FUNCTION_BLOCK B_SECCOM_CONTROLREMOTO (* Basic Function Block Type *)
  (* Standard: 61499-2 *)
  (* Version 0.0, 2015-12-09, 4DIAC-IDE, 4DIAC-Consortium *)
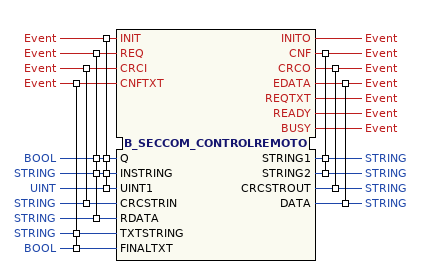
  EVENT_INPUT
    INIT WITH Q, UINT1, INSTRING; (* Initialization Request *)
    REQ WITH Q, INSTRING, RDATA; (* Normal Execution Request *)
    CRCI WITH CRCSTRIN;
    CNFTXT WITH TXTSTRING, FINALTXT;
  END_EVENT
  EVENT_OUTPUT
    INITO; (* Initialization Confirm *)
    CNF WITH STRING1, STRING2; (* Execution Confirmation *)
    CRCO WITH CRCSTROUT;
    EDATA WITH DATA;
    REQTXT;
    READY;
    BUSY;
  END_EVENT
  VAR_INPUT
    Q : BOOL; (* Input event qualifier *)
    INSTRING : STRING;
    UINT1 : UINT;
    CRCSTRIN : STRING;
    RDATA : STRING;
    TXTSTRING : STRING;
    FINALTXT : BOOL;
  END_VAR
  VAR_OUTPUT
    STRING1 : STRING;
    STRING2 : STRING;
    CRCSTROUT : STRING;
    DATA : STRING;
  END_VAR
  VAR
    STRSUB1 : STRING; (* Internal Variable *)
    STRSUB2 : STRING; (* Internal Variable *)
    STRSUB3 : STRING; (* Internal Variable *)
    INITCONTROL : BOOL := FALSE; (* Internal Variable *)
    UINTCPY : UINT := 0; (* Internal Variable *)
    LASTDLE : STRING; (* Internal Variable *)
    STRINGSPACE : STRING; (* Internal Variable *)
    SPACEINT : INT := 0; (* Internal Variable *)
    AUXINT1 : INT := 0; (* Internal Variable *)
    INTERNALVAR2 : BOOL; (* Internal Variable *)
  END_VAR
  EC_STATES
    START;
    State1 : start -> BUSY; (* Initial State *)
    SIMULACIONTECLADO : ST0 -> CNF;
    EJECUCIONPROGRAMA : EP0 -> CNF;
    PETICIONERRORES : PE0 -> CNF;
    LECTURAEJES : ST0 -> CNF;
    INFORMETIPO : ST0 -> CNF;
    ST1 : ST1 -> CRCO;
    ST2 : ST2 -> CNF;
    Exit_ST : -> READY;
    ST3 : ST3 -> CNF;
    ST4 : ST4 -> CNF;
    ST5 : ST5 -> CNF;
    INFOREESTADO : IE0 -> CNF;
    IE1 : IE1 -> CNF;
    IE2 : IE2 -> CNF;
    IE3 : IE3 -> CNF;
    IE4 : IE40 -> EDATA, IE4 -> CNF;
    Exit_IE : -> READY;
    InitEP : INIT -> CNF;
    InitPE : INIT -> CNF;
    Init_ST : INIT -> CNF;
    Init_LE : INIT -> CNF;
    Init_IT : INIT -> CNF;
    Init_IE : INIT -> CNF;
    PE1 : PE1 -> CRCO;
    PE2 : PE2 -> CNF;
    Exit_PE : -> READY;
    PE3 : PE3 -> CNF;
    PE4 : PE4 -> CNF;
    PE5 : PE50 -> EDATA, PE5 -> CNF;
    Exit_IT : -> READY;
    IT1 : IT1 -> CRCO;
    IT2 : ST2 -> CNF;
    IT3 : ST3 -> CNF;
    IT4 : ST4 -> CNF;
    IT5 : IT50 -> EDATA, ST5 -> CNF;
    Exit_LE : -> READY;
    LE1 : LE1 -> CRCO;
    LE2 : ST2 -> CNF;
    LE3 : ST3 -> CNF;
    LE4 : ST4 -> CNF;
    LE5 : LE50 -> EDATA, ST5 -> CNF;
    CARGAPROGRAMA : IE0 -> CNF;
    Exit_CP : -> READY;
    Init_CP : INIT -> CNF;
    CP1 : CP1 -> CRCO;
    CP4 : CP4 -> CRCO;
    CP2 : CP2 -> CNF;
    CP3 : -> REQTXT;
    CP6 : CP6 -> CNF;
    CP5 : CP5 -> CNF;
    EP1 : EP1 -> CRCO;
    EP2 : PE2 -> CNF;
    EP3 : PE3 -> CNF;
    Exit_PE_1 : -> READY;
    EP4 : PE4 -> CNF;
    EP5 : PE50 -> EDATA, PE5 -> CNF;
  END_STATES
  EC_TRANSITIONS
    SIMULACIONTECLADO TO ST1 := REQ&Q;
    ST1 TO ST2 := CRCI;
    SIMULACIONTECLADO TO Exit_ST := REQ&NOT Q;
    ST2 TO ST3 := REQ&Q;
    ST2 TO Exit_ST := REQ&NOT Q;
    ST3 TO ST4 := REQ&Q;
    ST4 TO ST5 := REQ&Q;
    ST3 TO Exit_ST := REQ&NOT Q;
    ST4 TO Exit_ST := REQ&NOT Q;
    ST5 TO Exit_ST := 1;
    INFOREESTADO TO IE1 := REQ&Q;
    IE1 TO IE2 := REQ&Q;
    IE2 TO IE3 := REQ&Q;
    IE3 TO IE4 := REQ&Q;
    INFOREESTADO TO Exit_IE := REQ&NOT Q;
    IE1 TO Exit_IE := REQ&NOT Q;
    IE2 TO Exit_IE := REQ&NOT Q;
    IE3 TO Exit_IE := REQ&NOT Q;
    IE4 TO Exit_IE := 1;
    State1 TO InitEP := UINTCPY=0 & INITCONTROL;
    InitEP TO EJECUCIONPROGRAMA := REQ&Q;
    InitPE TO PETICIONERRORES := REQ&Q;
    State1 TO InitPE := UINTCPY=1 & INITCONTROL;
    State1 TO Init_ST := UINTCPY=2 & INITCONTROL;
    State1 TO Init_LE := UINTCPY=3 & INITCONTROL;
    State1 TO Init_IT := UINTCPY=4 & INITCONTROL;
    State1 TO Init_IE := UINTCPY=5 & INITCONTROL;
    Init_ST TO SIMULACIONTECLADO := REQ&Q;
    Init_LE TO LECTURAEJES := REQ&Q;
    Init_IT TO INFORMETIPO := REQ&Q;
    Init_IE TO INFOREESTADO := REQ&Q;
    START TO State1 := INIT;
    Exit_IE TO START := 1;
    Exit_ST TO START := 1;
    State1 TO START := UINTCPY>6;
    PETICIONERRORES TO PE1 := REQ&Q;
    PE1 TO PE2 := CRCI;
    PE2 TO PE3 := REQ&Q;
    PE2 TO Exit_PE := REQ&NOT Q;
    PE3 TO Exit_PE := REQ&NOT Q;
    Exit_PE TO START := 1;
    PETICIONERRORES TO Exit_PE := REQ&NOT Q;
    PE3 TO PE4 := REQ&Q;
    PE4 TO PE5 := REQ&Q;
    PE4 TO Exit_PE := REQ&NOT Q;
    PE5 TO Exit_PE := 1;
    Exit_IT TO START := 1;
    IT1 TO IT2 := CRCI;
    INFORMETIPO TO IT1 := REQ&Q;
    IT2 TO IT3 := REQ&Q;
    IT3 TO IT4 := REQ&Q;
    IT4 TO IT5 := REQ&Q;
    IT1 TO Exit_IT := REQ&NOT Q;
    IT2 TO Exit_IT := REQ&NOT Q;
    IT3 TO Exit_IT := REQ&NOT Q;
    IT4 TO Exit_IT := REQ&NOT Q;
    IT5 TO Exit_IT := 1;
    INFORMETIPO TO Exit_IT := REQ&NOT Q;
    LECTURAEJES TO Exit_LE := REQ&NOT Q;
    Exit_LE TO START := 1;
    LECTURAEJES TO LE1 := REQ&Q;
    LE1 TO LE2 := CRCI;
    LE2 TO LE3 := REQ&Q;
    LE3 TO LE4 := REQ&Q;
    LE4 TO LE5 := REQ&Q;
    LE1 TO Exit_LE := REQ&NOT Q;
    LE2 TO Exit_LE := REQ&NOT Q;
    LE3 TO Exit_LE := REQ&NOT Q;
    LE4 TO Exit_LE := REQ&NOT Q;
    LE5 TO Exit_LE := 1;
    Init_CP TO CARGAPROGRAMA := REQ&Q;
    CARGAPROGRAMA TO Exit_CP := REQ&NOT Q;
    State1 TO Init_CP := UINTCPY=6 & INITCONTROL;
    Exit_CP TO START := 1;
    CARGAPROGRAMA TO CP1 := REQ&Q;
    CP1 TO CP2 := CRCI;
    CP2 TO CP3 := REQ&Q;
    CP3 TO CP4 := CNFTXT;
    CP4 TO CP5 := CRCI;
    CP5 TO CP3 := REQ&Q & NOT FINALTXT;
    CP5 TO CP6 := REQ&Q &  FINALTXT;
    CP6 TO Exit_CP := REQ;
    CP1 TO Exit_CP := REQ&NOT Q;
    CP2 TO Exit_CP := REQ&NOT Q;
    CP5 TO Exit_CP := REQ&NOT Q;
    EP1 TO EP2 := CRCI;
    EP2 TO EP3 := REQ&Q;
    EJECUCIONPROGRAMA TO Exit_PE_1 := REQ&NOT Q;
    EJECUCIONPROGRAMA TO EP1 := REQ&Q;
    EP3 TO EP4 := REQ&Q;
    EP4 TO EP5 := REQ&Q;
    EP2 TO Exit_PE_1 := REQ&NOT Q;
    EP3 TO Exit_PE_1 := REQ&NOT Q;
    EP4 TO Exit_PE_1 := REQ&NOT Q;
    EP5 TO Exit_PE_1 := 1;
    Exit_PE_1 TO START := 1;
  END_TRANSITIONS
  ALGORITHM INIT IN ST: (* Initialization algorithm *)
STRING1:='\x04\x7f';
STRING2:='\x01\x02\x03\x04';
INITCONTROL:=FALSE;
  END_ALGORITHM
  ALGORITHM REQ IN ST: (* Normally executed algorithm *)

  END_ALGORITHM
  ALGORITHM ST0 IN ST: (* new algorithm *)
STRING1:='\x05';
STRING2:='\x10\x30';
  END_ALGORITHM
  ALGORITHM ST1 IN ST: (* new algorithm *)
STRSUB1:='\x01\x52\x43\x4b\x02';
STRSUB2:='\x30\x32\x09';
STRSUB3:=CONCAT(STRSUB1,STRSUB2);

STRSUB2:=INSTRING;
STRSUB1:=CONCAT(STRSUB3,STRSUB2);

STRSUB2:='\x09\x03';
STRSUB3:=CONCAT(STRSUB1,STRSUB2);




CRCSTROUT:=STRSUB3;
  END_ALGORITHM
  ALGORITHM ST2 IN ST: (* new algorithm *)
STRING1:=CRCSTRIN;
STRING2:='\x10\x31';
  END_ALGORITHM
  ALGORITHM ST3 IN ST: (* new algorithm *)
STRING1:='\x04';
STRING2:='\x05\x7f';
  END_ALGORITHM
  ALGORITHM ST4 IN ST: (* new algorithm *)
STRING1:='\x10\x30';
STRING2:='\x02\x03';
  END_ALGORITHM
  ALGORITHM ST5 IN ST: (* new algorithm *)
STRING1:='\x10\x31';
STRING2:='\x04\x7f';
  END_ALGORITHM
  ALGORITHM EP0 IN ST: (* new algorithm *)
STRING1:='\x05';
STRING2:='\x10\x30';
  END_ALGORITHM
  ALGORITHM PE0 IN ST: (* new algorithm *)
STRING1:='\x05';
STRING2:='\x10\x30';
  END_ALGORITHM
  ALGORITHM LE0 IN ST: (* new algorithm *)
STRING1:='\x04\x33\x33\x7f';
STRING2:='\x01\x02\x03\x04';
  END_ALGORITHM
  ALGORITHM IT0 IN ST: (* new algorithm *)
STRING1:='\x04\x34\x34\x7f';
STRING2:='\x01\x02\x03\x04';
  END_ALGORITHM
  ALGORITHM IE0 IN ST: (* new algorithm *)
STRING1:='\x05';
STRING2:='\x10\x30';
  END_ALGORITHM
  ALGORITHM IE1 IN ST: (* new algorithm *)
STRING1:='\x01\x52\x43\x4c\x02\x03\xfe\x2c';
STRING2:='\x10\x31';
  END_ALGORITHM
  ALGORITHM IE2 IN ST: (* new algorithm *)
STRING1:='\x04';
STRING2:='\x05\x7f';
  END_ALGORITHM
  ALGORITHM IE3 IN ST: (* new algorithm *)
STRING1:='\x10\x30';
STRING2:='\x02\x03';
  END_ALGORITHM
  ALGORITHM IE4 IN ST: (* new algorithm *)
STRING1:='\x10\x31';
STRING2:='\x04\x7f';
  END_ALGORITHM
  ALGORITHM start IN ST: (* new algorithm *)
UINTCPY:=UINT1;
INITCONTROL:=TRUE;
  END_ALGORITHM
  ALGORITHM PE1 IN ST: (* new algorithm *)
STRSUB1:='\x01\x52\x43\x4b\x02';
STRSUB2:='\x30\x31';
STRSUB3:=CONCAT(STRSUB1,STRSUB2);

STRSUB2:='\x03';
STRSUB1:=CONCAT(STRSUB3,STRSUB2);

CRCSTROUT:=STRSUB1;
  END_ALGORITHM
  ALGORITHM PE2 IN ST: (* new algorithm *)
STRING1:=CRCSTRIN;
STRING2:='\x10\x31';
  END_ALGORITHM
  ALGORITHM PE3 IN ST: (* new algorithm *)
STRING1:='\x04';
STRING2:='\x05\x7f';
  END_ALGORITHM
  ALGORITHM PE4 IN ST: (* new algorithm *)
STRING1:='\x10\x30';
STRING2:='\x02\x03';
  END_ALGORITHM
  ALGORITHM PE5 IN ST: (* new algorithm *)
STRING1:='\x10\x31';
STRING2:='\x04\x7f';
  END_ALGORITHM
  ALGORITHM IT1 IN ST: (* new algorithm *)
STRSUB1:='\x01\x52\x43\x4b\x02';
STRSUB2:='\x31\x31';
STRSUB3:=CONCAT(STRSUB1,STRSUB2);

STRSUB2:='\x03';
STRSUB1:=CONCAT(STRSUB3,STRSUB2);

CRCSTROUT:=STRSUB1;
  END_ALGORITHM
  ALGORITHM LE1 IN ST: (* new algorithm *)
STRSUB1:='\x01\x52\x43\x4b\x02';
STRSUB2:='\x31\x30';
STRSUB3:=CONCAT(STRSUB1,STRSUB2);

STRSUB2:='\x03';
STRSUB1:=CONCAT(STRSUB3,STRSUB2);

CRCSTROUT:=STRSUB1;
  END_ALGORITHM
  ALGORITHM IE40 IN ST: (* new algorithm *)
DATA:=RDATA;
  END_ALGORITHM
  ALGORITHM IT50 IN ST: (* new algorithm *)
DATA:=RDATA;
  END_ALGORITHM
  ALGORITHM LE50 IN ST: (* new algorithm *)
DATA:=RDATA;
  END_ALGORITHM
  ALGORITHM PE50 IN ST: (* new algorithm *)
DATA:=RDATA;
  END_ALGORITHM
  ALGORITHM CP1 IN ST: (* new algorithm *)
STRSUB1:='\x01\x53\x43\x53\x02';
STRSUB2:='\x25\x36\x31\x34\x39\x39';
STRSUB3:=CONCAT(STRSUB1,STRSUB2);

STRSUB2:='\x09\x44';
STRSUB1:=CONCAT(STRSUB3,STRSUB2);

STRSUB2:='\x17';
STRSUB3:=CONCAT(STRSUB1,STRSUB2);

CRCSTROUT:=STRSUB3;
  END_ALGORITHM
  ALGORITHM CP2 IN ST: (* new algorithm *)
STRING1:=CRCSTRIN;
LASTDLE:='\x10\x31';
STRING2:='\x10\x31';
  END_ALGORITHM
  ALGORITHM CP4 IN ST: (* new algorithm *)
STRSUB1:='\x02';
STRSUB2:=TXTSTRING;
STRINGSPACE:='\x20';

SPACEINT:=0;
AUXINT1:=LEN(STRSUB2);
WHILE SPACEINT<=AUXINT1 DO
	STRSUB3:=MID(STRSUB2,1,SPACEINT);
	IF STRSUB3=STRINGSPACE THEN
		STRSUB2:=DELETE(STRSUB2,1,SPACEINT);
		AUXINT1:=LEN(STRSUB2);
	ELSE
	SPACEINT:=SPACEINT+1;

	END_IF;

END_WHILE;

STRSUB3:=CONCAT(STRSUB1,STRSUB2);

IF FINALTXT=TRUE THEN
	STRSUB2:='\x03';
ELSE
	STRSUB2:='\x17';
END_IF;

STRSUB1:=CONCAT(STRSUB3,STRSUB2);

CRCSTROUT:=STRSUB1;
  END_ALGORITHM
  ALGORITHM CP5 IN ST: (* new algorithm *)
STRING1:=CRCSTRIN;

IF LASTDLE='\x10\x30' THEN
STRING2:='\x10\x31';
LASTDLE:='\x10\x31';
ELSE
STRING2:='\x10\x30';
LASTDLE:='\x10\x30';
END_IF;
  END_ALGORITHM
  ALGORITHM CP6 IN ST: (* new algorithm *)
STRING1:='\x04';
STRING2:='\x01\x02\x03\x04';
  END_ALGORITHM
  ALGORITHM EP1 IN ST: (* new algorithm *)
STRSUB1:='\x01\x52\x43\x4b\x02';
STRSUB2:='\x30\x30';
STRSUB3:=CONCAT(STRSUB1,STRSUB2);

STRSUB2:='\x25\x36\x31\x34\x39\x39\x4e\x30\x30\x30\x30\x03';
STRSUB1:=CONCAT(STRSUB3,STRSUB2);

CRCSTROUT:=STRSUB1;
  END_ALGORITHM
END_FUNCTION_BLOCK
